// TIA Portal V14 SP1 export
// export: Created 2019-04-23T05:55:13.4851404Z, ExportSetting WithDefaults, WithReadOnly, DisplayName Totally Integrated Automation Portal, DisplayVersion V14 SP1 Update 6, DisplayName TIA Portal Openness, DisplayVersion V14 SP1 Update 6, DisplayName STEP 7 Professional, DisplayVersion V14 SP1 Update 6, DisplayName WinCC Professional, DisplayVersion V14 SP1 Update 6
FUNCTION_BLOCK "453UF_Invertor"   // FB2031, LAD
TITLE = Блок управления инвертором 111UF
{ S7_Optimized_Access := 'FALSE' }
VERSION : 0.1
// stored: AutoNumber false, CodeModifiedDate 2019-03-26T07:08:56.819049Z, CompileDate 2019-03-26T07:08:56.8434631Z, CreationDate 2019-02-26T05:18:41.6523018Z, InterfaceModifiedDate 2019-01-10T08:54:25.4366574Z, IsConsistent true, IsIECCheckEnabled false, IsKnowHowProtected false, ISMultiInstanceCapable true, IsWriteProtected false, LibraryConformanceStatus Warning: The object contains access to global data blocks. Warning: The block contains direct access to inputs, outputs, bit memories, indirect access to the registry or indirect access to external memory areas that are unknown at the time of compilation., ModifiedDate 2019-03-26T07:08:56.819049Z, ParameterModified 2018-11-15T11:45:53.3082246Z, StructureModified 2019-01-10T08:54:25.4366574Z, UDAEnableTagReadback false
   VAR DB_SPECIFIC
      HMI : Struct
         CMD : Struct
            Start : Bool;   // Команда старта вибратора / Команда старт вращения
            Stop : Bool;   // Команда останова вибратора / Команда стоп вращения
            Spare_2 : Bool;
            Spare_3 : Bool;
            Spare_4 : Bool;
            Spare_5 : Bool;
            Manual : Bool;   // Ручной режим управления
            Reset_Error : Bool;   // Сброс ошибок
         END_STRUCT;
         DATA : Struct
            StatusWord : Word;   // Слово состояния блока управления
            Ref_Speed_Invertor : Real;   // Значение скорости задаваемое на инвертор
            Wait_Time : DInt := 5;   // Время контроля включения реле / Время задержки старта инвертора (*100msec)
            Man_Ref_Speed : Real := 20.0;   // Скорость вращения в ручном режиме (Гц)
            Max_Invert_Speed : Real := 50.0;   // Максимальная частота инвертора
            Overflow_Sensor_Time : DInt := 2;   // Время контроля включения реле / Время задержки опроса датчика переполнения шнека (*100msec)
            Sensor_Overflow_Not_OK : Bool;   // Сработал датчик переполнения шнека
            Max_Lvl_RotorFider_Bunker : Bool;   // Максимальный уровень смеси в накопителе роторного питателя подачи в силосы смеси
            Stop_Max_Lvl_RotorFider_Bunker : Bool;   // Останов подачи смеси в накопитель по причине переполнения накопителя роторн. питателя
            Spare_10 : Bool;
            Spare_9 : Bool;
            Spare_8 : Bool;
            Spare_7 : Bool;
            Spare_6 : Bool;
            Auto_Ref_Speed_Fast : Real := 15.0;   // Скорость вращения быстро в автом. режиме (Гц)
            Auto_Ref_Speed_Slow : Real := 35.0;   // Скорость вращения медленно в автом. режиме (Гц)
            Max_Lvl_RotorFider_Bunker_Time : DInt := 5;   // Время задержки опроса датчика переполнения накопителя роторного питателя (sec)
         END_STRUCT;
      END_STRUCT;
   END_VAR
   VAR
      Inverter : "Menage_Analog_Inverter";   // Блок управления инвертором
      Ramp : "Ramp_Calc";   // Блок формирования рампы привода
      TimerDriveStart : TON;
      TimerOverflow_Sensor : TON;
      Bunker_Time : TON;
      Stop_Timer : TON;
   END_VAR
   VAR DB_SPECIFIC
      Ramp_SpdSet : Real;   // Задание скорости перемещения на блок обработки рампы
      SpeedRampOut : Real;   // Значение скорости перемещения после блока рампы
      Wait_Time : Time;   // Время контроля включения реле / Время задержки старта инвертора
      Overflow_Sensor_Time : Time;   // Время задержки опроса датчика переполнения
      Max_Lvl_RotorFider_Bunker_Time : Time;   // Время задержки опроса датчика переполнения накопителя роторного питателя
      ResetErr : Bool;   // Сброс ошибок блока управления
      General_cond_OK : Bool;   // Выполнены условия разрешения работы механизма
      ManCmd_MoveFwd : Bool;   // Наличие команды на вращение вперёд в ручном
      Manual_Mode : Bool;   // Ручной режим управления
      AutoCmd_MoveFast : Bool;   // Наличие команды на вращение вперёд в автомате быстрая скорость
      AutoCmd_MoveSlow : Bool;   // Наличие команды на вращение назад в автомате медленная скорость
      Sensor_Overflow_Not_OK : Bool;   // Сработал датчик переполнения
      DriveStart : Bool;   // Команда разрешения работы привода
      DriveEnable : Bool;   // Команда на включение привода
      Motor_ON : Bool;   // Наличие подключенного мотора к инвертору
      Cmd_Man_ON : Bool;   // Наличие команды вращения в ручном режиме
      Stop_Max_Lvl_RotorFider_Bunker : Bool;   // Останов подачи смеси в накопитель
      Spare : Bool;
      Spare_4 : Bool;
      Spare_3 : Bool;
      Spare_2 : Bool;
   END_VAR
   VAR_TEMP
      Temp_INT : Int;
      Temp_Bit : Bool;
   END_VAR
   VAR_TEMP   // added for the SCL form of the ladder/FBD networks
      _w1 : Bool;
   END_VAR
BEGIN

REGION Network 2: Проверка готовности аварийных систем / Ïðîâåðêà ñîñòîÿíèÿ ýëåêòðè÷åñêèõ öåïåé
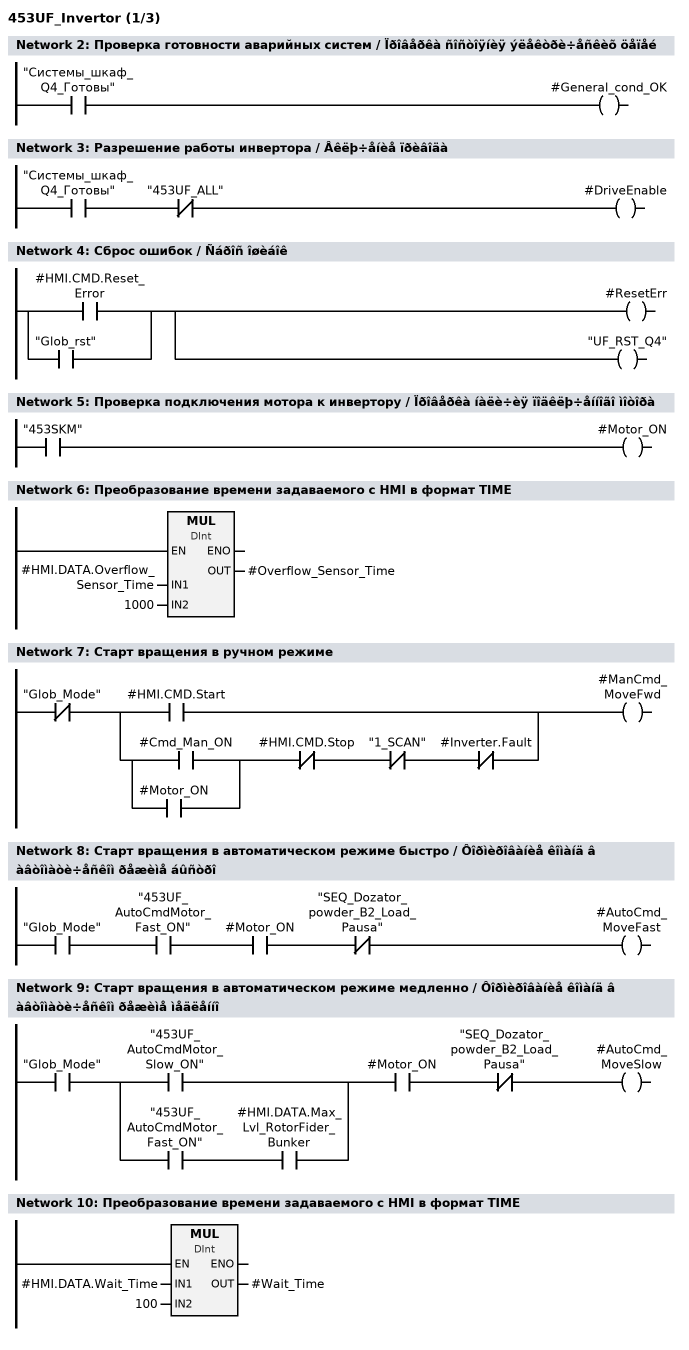
   RUNG wire#powerrail
      Contact( "Системы_шкаф_Q4_Готовы" )
      Coil( #General_cond_OK )
   END_RUNG
   // the same network as SCL:
   #General_cond_OK := "Системы_шкаф_Q4_Готовы";
END_REGION

REGION Network 3: Разрешение работы инвертора / Âêëþ÷åíèå ïðèâîäà
   RUNG wire#powerrail
      Contact( "Системы_шкаф_Q4_Готовы" )
      I_Contact( "453UF_ALL" )
      Coil( #DriveEnable )
   END_RUNG
   // the same network as SCL:
   #DriveEnable := "Системы_шкаф_Q4_Готовы" AND NOT "453UF_ALL";
END_REGION

REGION Network 4: Сброс ошибок / Ñáðîñ îøèáîê
   RUNG wire#powerrail
      Contact( #HMI.CMD.Reset_Error )
      wire#w1
      Coil( #ResetErr )
   END_RUNG
   RUNG wire#powerrail
      Contact( "Glob_rst" )
   END_RUNG wire#w1
   RUNG wire#w1
      Coil( "UF_RST_Q4" )
   END_RUNG
   // the same network as SCL:
   #ResetErr := #HMI.CMD.Reset_Error OR "Glob_rst";
   "UF_RST_Q4" := #ResetErr;
END_REGION

REGION Network 5: Проверка подключения мотора к инвертору / Ïðîâåðêà íàëè÷èÿ ïîäêëþ÷åííîãî ìîòîðà
   RUNG wire#powerrail
      Contact( "453SKM" )
      Coil( #Motor_ON )
   END_RUNG
   // the same network as SCL:
   #Motor_ON := "453SKM";
END_REGION

REGION Network 6: Преобразование времени задаваемого с HMI в формат TIME
   RUNG wire#powerrail
      { S7_Templates := "SrcType := DInt"; S7_GenerateENO := "TRUE" } Mul(in1 := #HMI.DATA.Overflow_Sensor_Time, in2 := 1000, out => #Overflow_Sensor_Time)
   END_RUNG
   // the same network as SCL:
   #Overflow_Sensor_Time := #HMI.DATA.Overflow_Sensor_Time * 1000;
END_REGION

REGION Network 7: Старт вращения в ручном режиме
   RUNG wire#powerrail
      I_Contact( "Glob_Mode" )
      wire#w1
      Contact( #HMI.CMD.Start )
      wire#w2
      Coil( #ManCmd_MoveFwd )
   END_RUNG
   RUNG wire#w1
      Contact( #Cmd_Man_ON )
      wire#w3
      I_Contact( #HMI.CMD.Stop )
      I_Contact( "1_SCAN" )
      I_Contact( #Inverter.Fault )
   END_RUNG wire#w2
   RUNG wire#w1
      Contact( #Motor_ON )
   END_RUNG wire#w3
   // the same network as SCL:
   #ManCmd_MoveFwd := NOT "Glob_Mode" AND (#HMI.CMD.Start OR ((#Cmd_Man_ON OR #Motor_ON) AND NOT #HMI.CMD.Stop AND NOT "1_SCAN" AND NOT #Inverter.Fault));
END_REGION

REGION Network 8: Старт вращения в автоматическом режиме быстро / Ôîðìèðîâàíèå êîìàíä â àâòîìàòè÷åñêîì ðåæèìå áûñòðî
   RUNG wire#powerrail
      Contact( "Glob_Mode" )
      Contact( "453UF_AutoCmdMotor_Fast_ON" )
      Contact( #Motor_ON )
      I_Contact( "SEQ_Dozator_powder_B2_Load_Pausa" )
      Coil( #AutoCmd_MoveFast )
   END_RUNG
   // the same network as SCL:
   #AutoCmd_MoveFast := "Glob_Mode" AND "453UF_AutoCmdMotor_Fast_ON" AND #Motor_ON AND NOT "SEQ_Dozator_powder_B2_Load_Pausa";
END_REGION

REGION Network 9: Старт вращения в автоматическом режиме медленно / Ôîðìèðîâàíèå êîìàíä â àâòîìàòè÷åñêîì ðåæèìå ìåäëåííî
   RUNG wire#powerrail
      Contact( "Glob_Mode" )
      wire#w1
      Contact( "453UF_AutoCmdMotor_Slow_ON" )
      wire#w2
      Contact( #Motor_ON )
      I_Contact( "SEQ_Dozator_powder_B2_Load_Pausa" )
      Coil( #AutoCmd_MoveSlow )
   END_RUNG
   RUNG wire#w1
      Contact( "453UF_AutoCmdMotor_Fast_ON" )
      Contact( #HMI.DATA.Max_Lvl_RotorFider_Bunker )
   END_RUNG wire#w2
   // the same network as SCL:
   #AutoCmd_MoveSlow := "Glob_Mode" AND ("453UF_AutoCmdMotor_Slow_ON" OR ("453UF_AutoCmdMotor_Fast_ON" AND #HMI.DATA.Max_Lvl_RotorFider_Bunker)) AND #Motor_ON AND NOT "SEQ_Dozator_powder_B2_Load_Pausa";
END_REGION

REGION Network 10: Преобразование времени задаваемого с HMI в формат TIME
   RUNG wire#powerrail
      { S7_Templates := "SrcType := DInt"; S7_GenerateENO := "TRUE" } Mul(in1 := #HMI.DATA.Wait_Time, in2 := 100, out => #Wait_Time)
   END_RUNG
   // the same network as SCL:
   #Wait_Time := #HMI.DATA.Wait_Time * 100;
END_REGION

REGION Network 11: Формирование команды RUN для инвертора / Ôîðìèðîâàíèå êîìàíäû ñòàðòà ðàáîòû èíâåðòîðà
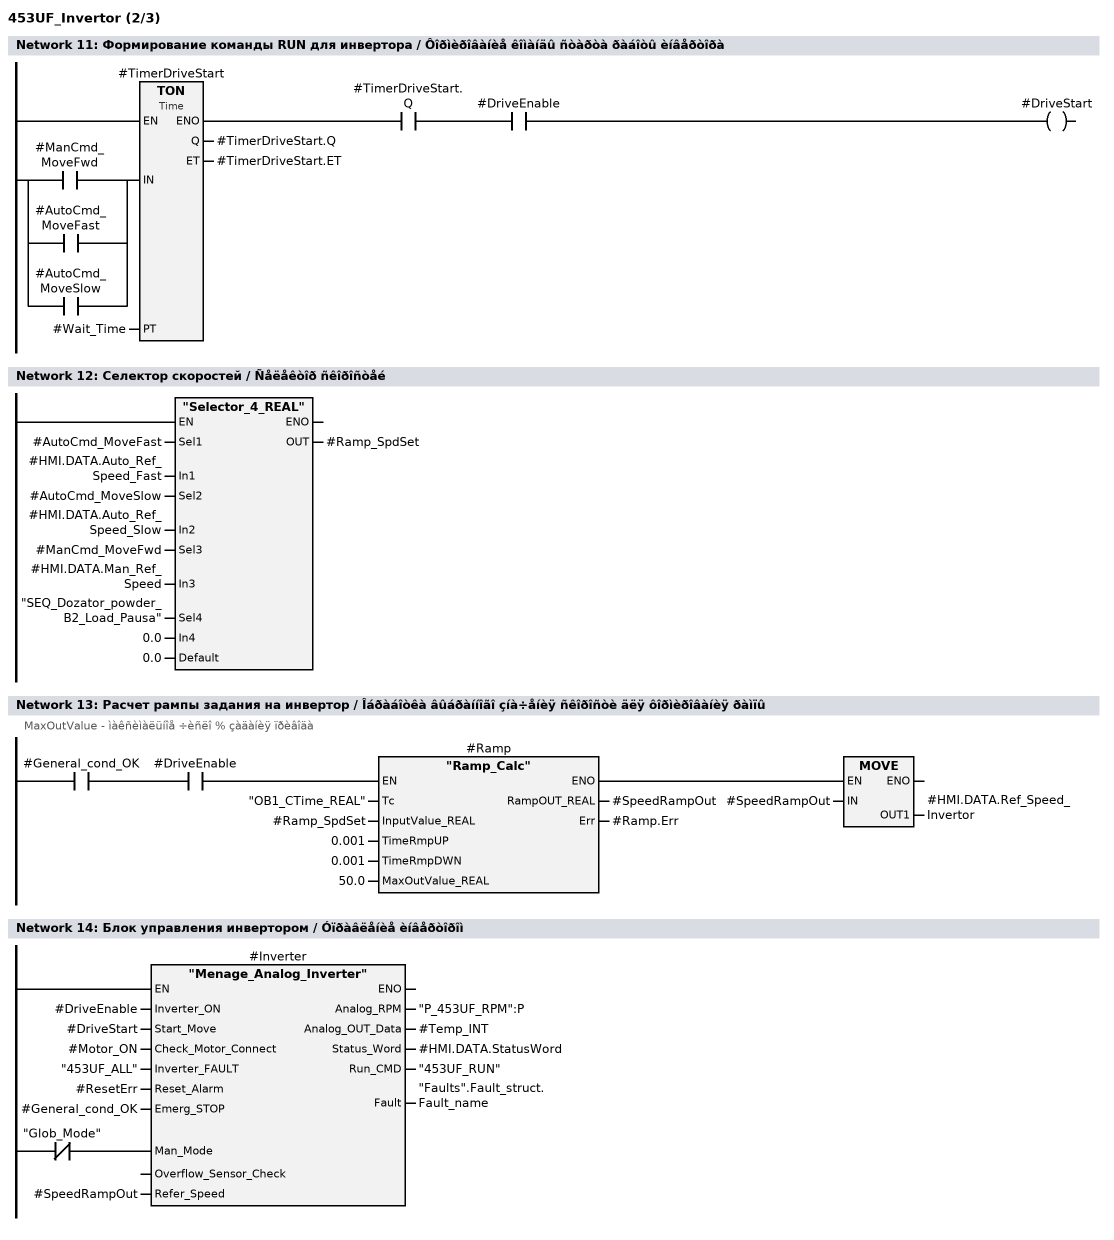
   #TimerDriveStart.TON(IN := #ManCmd_MoveFwd OR #AutoCmd_MoveFast OR #AutoCmd_MoveSlow,
                        PT := #Wait_Time,
                        Q => #TimerDriveStart.Q,
                        ET => #TimerDriveStart.ET,
                        ENO => #_w1);
   #DriveStart := #_w1 AND #TimerDriveStart.Q AND #DriveEnable;
END_REGION

REGION Network 12: Селектор скоростей / Ñåëåêòîð ñêîðîñòåé
   RUNG wire#powerrail
      "Selector_4_REAL"(Sel1 := #AutoCmd_MoveFast, In1 := #HMI.DATA.Auto_Ref_Speed_Fast, Sel2 := #AutoCmd_MoveSlow, In2 := #HMI.DATA.Auto_Ref_Speed_Slow, Sel3 := #ManCmd_MoveFwd, In3 := #HMI.DATA.Man_Ref_Speed, Sel4 := "SEQ_Dozator_powder_B2_Load_Pausa", In4 := 0.0, Default := 0.0, OUT => #Ramp_SpdSet)
   END_RUNG
   // the same network as SCL:
   "Selector_4_REAL"(Sel1 := #AutoCmd_MoveFast,
                     In1 := #HMI.DATA.Auto_Ref_Speed_Fast,
                     Sel2 := #AutoCmd_MoveSlow,
                     In2 := #HMI.DATA.Auto_Ref_Speed_Slow,
                     Sel3 := #ManCmd_MoveFwd,
                     In3 := #HMI.DATA.Man_Ref_Speed,
                     Sel4 := "SEQ_Dozator_powder_B2_Load_Pausa",
                     In4 := 0.0,
                     Default := 0.0,
                     OUT => #Ramp_SpdSet);
END_REGION

REGION Network 13: Расчет рампы задания на инвертор / Îáðàáîòêà âûáðàííîãî çíà÷åíèÿ ñêîðîñòè äëÿ ôîðìèðîâàíèÿ ðàìïû
   // MaxOutValue - ìàêñèìàëüíîå ÷èñëî % çàäàíèÿ ïðèâîäà
   RUNG wire#powerrail
      Contact( #General_cond_OK )
      Contact( #DriveEnable )
      #Ramp(Tc := "OB1_CTime_REAL", InputValue_REAL := #Ramp_SpdSet, TimeRmpUP := 0.001, TimeRmpDWN := 0.001, MaxOutValue_REAL := 50.0, RampOUT_REAL => #SpeedRampOut, Err => #Ramp.Err)
      { S7_GenerateENO := "TRUE" } Move(in := #SpeedRampOut, out1 => #HMI.DATA.Ref_Speed_Invertor)
   END_RUNG
   // the same network as SCL:
   #Ramp(EN := #General_cond_OK AND #DriveEnable,   // "Ramp_Calc"
         Tc := "OB1_CTime_REAL",
         InputValue_REAL := #Ramp_SpdSet,
         TimeRmpUP := 0.001,
         TimeRmpDWN := 0.001,
         MaxOutValue_REAL := 50.0,
         RampOUT_REAL => #SpeedRampOut,
         Err => #Ramp.Err,
         ENO => #_w1);
   IF #_w1 THEN #HMI.DATA.Ref_Speed_Invertor := #SpeedRampOut; END_IF;
END_REGION

REGION Network 14: Блок управления инвертором / Óïðàâëåíèå èíâåðòîðîì
   RUNG wire#powerrail
      #Inverter(Man_Mode := wire#w1, Inverter_ON := #DriveEnable, Start_Move := #DriveStart, Check_Motor_Connect := #Motor_ON, Inverter_FAULT := "453UF_ALL", Reset_Alarm := #ResetErr, Emerg_STOP := #General_cond_OK, Overflow_Sensor_Check :=, Refer_Speed := #SpeedRampOut, Analog_RPM => "P_453UF_RPM":P, Analog_OUT_Data => #Temp_INT, Status_Word => #HMI.DATA.StatusWord, Run_CMD => "453UF_RUN", Fault => "Faults".Fault_struct.Fault_name)
   END_RUNG
   RUNG wire#powerrail
      I_Contact( "Glob_Mode" )
   END_RUNG wire#w1
   // the same network as SCL:
   #Inverter(Inverter_ON := #DriveEnable,   // "Menage_Analog_Inverter"
             Start_Move := #DriveStart,
             Check_Motor_Connect := #Motor_ON,
             Inverter_FAULT := "453UF_ALL",
             Reset_Alarm := #ResetErr,
             Emerg_STOP := #General_cond_OK,
             Man_Mode := NOT "Glob_Mode",
             Refer_Speed := #SpeedRampOut,
             Analog_RPM => "P_453UF_RPM":P,
             Analog_OUT_Data => #Temp_INT,
             Status_Word => #HMI.DATA.StatusWord,
             Run_CMD => "453UF_RUN",
             Fault => "Faults".Fault_struct.Fault_name);
END_REGION

REGION Network 15: Преобразование времени задаваемого с HMI в формат TIME
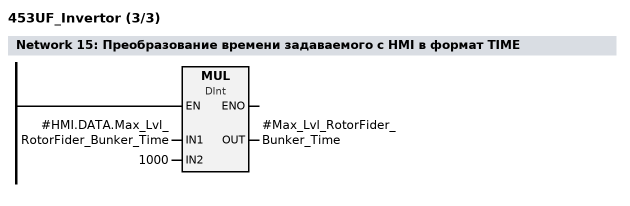
   RUNG wire#powerrail
      { S7_Templates := "SrcType := DInt"; S7_GenerateENO := "TRUE" } Mul(in1 := #HMI.DATA.Max_Lvl_RotorFider_Bunker_Time, in2 := 1000, out => #Max_Lvl_RotorFider_Bunker_Time)
   END_RUNG
   // the same network as SCL:
   #Max_Lvl_RotorFider_Bunker_Time := #HMI.DATA.Max_Lvl_RotorFider_Bunker_Time * 1000;
END_REGION
END_FUNCTION_BLOCK
